PROGRAM PTab_Out

VAR_INPUT
	fPwmInput								: FLOAT;	
END_VAR

VAR
	bPwmOutBitPos							: BOOL;
	bPwmOutBitNeg							: BOOL;

	fbCTRL_PWM_OUT							: FB_CTRL_PWM_OUT;
	stCTRL_PWM_OUT_PARAMS					: ST_CTRL_PWM_OUT_PARAMS;

	eMode									: E_CTRL_MODE;
	eErrorId								: E_CTRL_ERRORCODES;
	bError									: BOOL;

	bInit									: BOOL		:= TRUE;
	fDelta									: FLOAT	:= 0.05;
END_VAR

IF bInit
THEN
	(* Init parameter struct *)
	stCTRL_PWM_OUT_PARAMS.tTaskCycleTime	:= T#10MS;
	stCTRL_PWM_OUT_PARAMS.tPWMPeriod		:= T#200MS;

	(* ACTIVE --> normal operation *)
	eMode									:= eCTRL_MODE_ACTIVE;

	(* Reset the init flag *)
	bInit									:= FALSE;
END_IF

fbCTRL_PWM_OUT(		fPwmInput				:= fPwmInput,
							eMode			:= eMode,
							stParams		:= stCTRL_PWM_OUT_PARAMS,
							
							bPwmOutBitPos	=> bPwmOutBitPos,
							bPwmOutBitNeg	=> bPwmOutBitNeg,
							bError			=> bError,
							eErrorId		=> eErrorId
						);
						
	(* Output sign   *)
IOS.IO_Out_Aque_Mesa:=bPwmOutBitPos;

END_PROGRAM

(* stored: Version 1.1.0.1, ProductVersion 3.1.4020.12
   POU PTab_Out: Id {97dc895a-311f-4097-8c38-c3fc67b0baaf}, SpecialFunc None *)
